// TIA Portal project "GirelloAutomatico_Curto_Claudio" (V15.1)

(* hardware
DEVICE "S7-1200 station_1"  S7-1200 Station
   slot 0: "Telaio di montaggio_0"  S7-1200 Rack  Rack  V1.0
   slot 1: "PLC_1"  CPU 1214C DC/DC/DC  6ES7 214-1AG40-0XB0  V4.2
*)

// ===== PLC "PLC_1"  CPU 1214C DC/DC/DC =====

VAR_GLOBAL   // PLC tag table "Tabella delle variabili standard"
   "P1" AT %I0.0 : Bool;
   "P2" AT %I0.1 : Bool;
   "PG" AT %I0.2 : Bool;
   "PX" AT %I0.3 : Bool;
   "FCS" AT %I0.4 : Bool;
   "FCD" AT %I0.5 : Bool;
   "M1" AT %Q0.0 : Bool;
   "M2" AT %Q0.1 : Bool;
   "MG" AT %Q0.2 : Bool;
   "S" AT %Q0.3 : Bool;
   "D" AT %Q0.4 : Bool;
END_VAR

DATA_BLOCK "VariabiliStato"   // DB1
{ S7_Optimized_Access := 'TRUE' }
VERSION : 0.1
   VAR RETAIN
      Home : Bool := true;
   END_VAR
   VAR
      Muovi_1 : Bool;
      Muovi_MG : Bool;
      Ruota_S : Bool;
      Muovi_2 : Bool;
      Ruota_D : Bool;
   END_VAR
BEGIN
END_DATA_BLOCK

ORGANIZATION_BLOCK "Main"   // OB1, LAD, ProgramCycle
TITLE = "Main Program Sweep (Cycle)"
{ S7_Optimized_Access := 'TRUE' }
VERSION : 0.1
   VAR_INPUT
      Initial_Call : Bool;   // Initial call of this OB
      Remanence : Bool;   // =True, if remanent data are available
   END_VAR
BEGIN

REGION Network 1
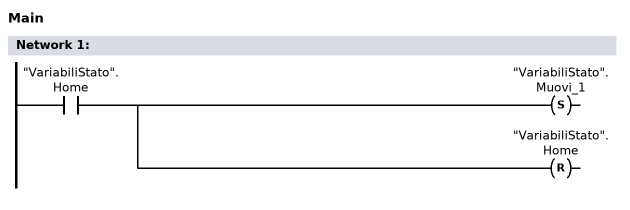
   RUNG wire#powerrail
      Contact( "VariabiliStato".Home )
      wire#w1
      S_Coil( "VariabiliStato".Muovi_1 )
   END_RUNG
   RUNG wire#w1
      R_Coil( "VariabiliStato".Home )
   END_RUNG
   // the same network as SCL:
   IF "VariabiliStato".Home THEN
       "VariabiliStato".Muovi_1 := TRUE;
       "VariabiliStato".Home := FALSE;
   END_IF;
END_REGION
END_ORGANIZATION_BLOCK

ORGANIZATION_BLOCK "Nastro_1"   // OB123, LAD, ProgramCycle
TITLE = "Main Program Sweep (Cycle)"
{ S7_Optimized_Access := 'TRUE' }
VERSION : 0.1
   VAR_INPUT
      Initial_Call : Bool;   // Initial call of this OB
      Remanence : Bool;   // =True, if remanent data are available
   END_VAR
BEGIN

REGION Network 1
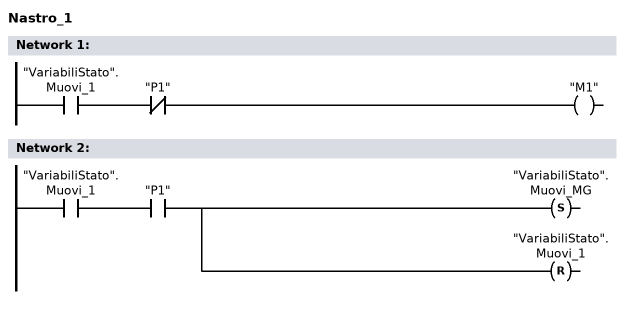
   RUNG wire#powerrail
      Contact( "VariabiliStato".Muovi_1 )
      I_Contact( "P1" )
      Coil( "M1" )
   END_RUNG
   // the same network as SCL:
   "M1" := "VariabiliStato".Muovi_1 AND NOT "P1";
END_REGION

REGION Network 2
   RUNG wire#powerrail
      Contact( "VariabiliStato".Muovi_1 )
      Contact( "P1" )
      wire#w1
      S_Coil( "VariabiliStato".Muovi_MG )
   END_RUNG
   RUNG wire#w1
      R_Coil( "VariabiliStato".Muovi_1 )
   END_RUNG
   // the same network as SCL:
   IF "VariabiliStato".Muovi_1 AND "P1" THEN
       "VariabiliStato".Muovi_MG := TRUE;
       "VariabiliStato".Muovi_1 := FALSE;
   END_IF;
END_REGION
END_ORGANIZATION_BLOCK

ORGANIZATION_BLOCK "Girello"   // OB124, LAD, ProgramCycle
TITLE = "Main Program Sweep (Cycle)"
{ S7_Optimized_Access := 'TRUE' }
VERSION : 0.1
   VAR_INPUT
      Initial_Call : Bool;   // Initial call of this OB
      Remanence : Bool;   // =True, if remanent data are available
   END_VAR
BEGIN

REGION Network 1
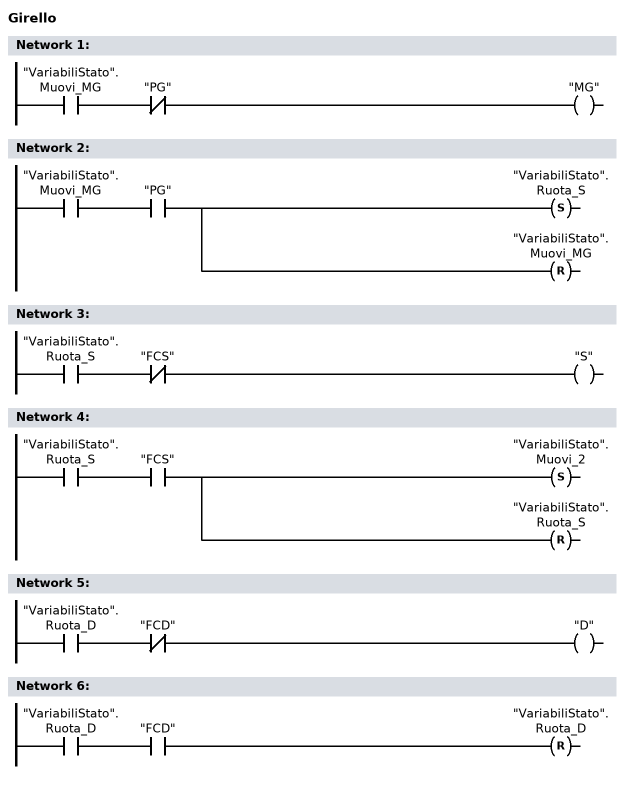
   RUNG wire#powerrail
      Contact( "VariabiliStato".Muovi_MG )
      I_Contact( "PG" )
      Coil( "MG" )
   END_RUNG
   // the same network as SCL:
   "MG" := "VariabiliStato".Muovi_MG AND NOT "PG";
END_REGION

REGION Network 2
   RUNG wire#powerrail
      Contact( "VariabiliStato".Muovi_MG )
      Contact( "PG" )
      wire#w1
      S_Coil( "VariabiliStato".Ruota_S )
   END_RUNG
   RUNG wire#w1
      R_Coil( "VariabiliStato".Muovi_MG )
   END_RUNG
   // the same network as SCL:
   IF "VariabiliStato".Muovi_MG AND "PG" THEN
       "VariabiliStato".Ruota_S := TRUE;
       "VariabiliStato".Muovi_MG := FALSE;
   END_IF;
END_REGION

REGION Network 3
   RUNG wire#powerrail
      Contact( "VariabiliStato".Ruota_S )
      I_Contact( "FCS" )
      Coil( "S" )
   END_RUNG
   // the same network as SCL:
   "S" := "VariabiliStato".Ruota_S AND NOT "FCS";
END_REGION

REGION Network 4
   RUNG wire#powerrail
      Contact( "VariabiliStato".Ruota_S )
      Contact( "FCS" )
      wire#w1
      S_Coil( "VariabiliStato".Muovi_2 )
   END_RUNG
   RUNG wire#w1
      R_Coil( "VariabiliStato".Ruota_S )
   END_RUNG
   // the same network as SCL:
   IF "VariabiliStato".Ruota_S AND "FCS" THEN
       "VariabiliStato".Muovi_2 := TRUE;
       "VariabiliStato".Ruota_S := FALSE;
   END_IF;
END_REGION

REGION Network 5
   RUNG wire#powerrail
      Contact( "VariabiliStato".Ruota_D )
      I_Contact( "FCD" )
      Coil( "D" )
   END_RUNG
   // the same network as SCL:
   "D" := "VariabiliStato".Ruota_D AND NOT "FCD";
END_REGION

REGION Network 6
   RUNG wire#powerrail
      Contact( "VariabiliStato".Ruota_D )
      Contact( "FCD" )
      R_Coil( "VariabiliStato".Ruota_D )
   END_RUNG
   // the same network as SCL:
   IF "VariabiliStato".Ruota_D AND "FCD" THEN "VariabiliStato".Ruota_D := FALSE; END_IF;
END_REGION
END_ORGANIZATION_BLOCK

ORGANIZATION_BLOCK "Nastro_2"   // OB125, LAD, ProgramCycle
TITLE = "Main Program Sweep (Cycle)"
{ S7_Optimized_Access := 'TRUE' }
VERSION : 0.1
   VAR_INPUT
      Initial_Call : Bool;   // Initial call of this OB
      Remanence : Bool;   // =True, if remanent data are available
   END_VAR
BEGIN

REGION Network 1
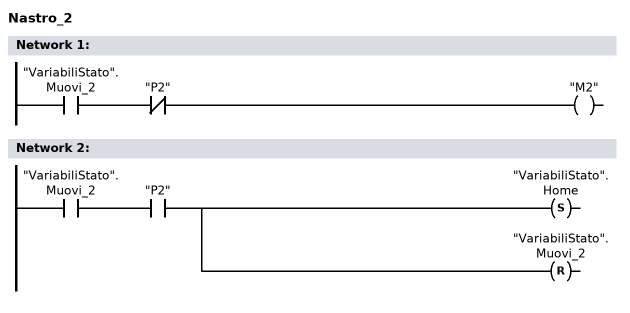
   RUNG wire#powerrail
      Contact( "VariabiliStato".Muovi_2 )
      I_Contact( "P2" )
      Coil( "M2" )
   END_RUNG
   // the same network as SCL:
   "M2" := "VariabiliStato".Muovi_2 AND NOT "P2";
END_REGION

REGION Network 2
   RUNG wire#powerrail
      Contact( "VariabiliStato".Muovi_2 )
      Contact( "P2" )
      wire#w1
      S_Coil( "VariabiliStato".Home )
   END_RUNG
   RUNG wire#w1
      R_Coil( "VariabiliStato".Muovi_2 )
   END_RUNG
   // the same network as SCL:
   IF "VariabiliStato".Muovi_2 AND "P2" THEN
       "VariabiliStato".Home := TRUE;
       "VariabiliStato".Muovi_2 := FALSE;
   END_IF;
END_REGION
END_ORGANIZATION_BLOCK